// TIA Portal V17 export
// export: Created 2025-03-05T08:02:19.8399003Z, ExportSetting WithDefaults, DisplayName Totally Integrated Automation Portal, DisplayVersion V17 Update 8, DisplayName TIA Portal Openness, DisplayVersion V17 Update 8, DisplayName TIA Portal Version Control Interface, DisplayVersion V17, DisplayName SINAMICS Startdrive Advanced, DisplayVersion V17 SP2, DisplayName SINAMICS Startdrive G110M, G120, G120C, G120D, G120P, G115D, DisplayVersion V17 SP2, DisplayName SINAMICS Startdrive G130, G150, S120, S150, SINAMICS MV, S210, DisplayVersion V17 SP2, DisplayName STEP 7 Professional, DisplayVersion V17 Update 8, DisplayName SINUMERIK ONE STEP 7 Toolbox, DisplayVersion V17 Update 12, DisplayName SINUMERIK 840D sl STEP 7 Toolbox, DisplayVersion V17 Update 12, DisplayName STEP 7 Safety, DisplayVersion V17 Update 6, DisplayName WinCC Advanced, DisplayVersion V17 Update 8
TYPE "AXIS_MANAGEMENT"
// stored: IsFailsafeCompliant false
   STRUCT
      UNIT_01_HM_PSTN : Bool;   // UNIT 01 HOME POSITION
      UNIT_01_MAINT_POS : Bool;   // UNIT 01 MAINTENACE POSITION
      UNIT_01_ST1_OUT_OF_CLLSN_ST0 : Bool;   // UNIT 01 STATION 1 OUT OF COLLISION STATION 0
      UNIT_01_ST2_OUT_OF_CLLSN_ST0 : Bool;   // UNIT 01 STATION 2 OUT OF COLLISION STATION 0
      UNIT_01_ST3_OUT_OF_CLLSN_ST0 : Bool;   // UNIT 01 STATION 3 OUT OF COLLISION STATION 0
      UNIT_01_ST4_OUT_OF_CLLSN_ST0 : Bool;   // UNIT 01 STATION 4 OUT OF COLLISION STATION 0
      UNIT_01_ST3_AX_IN_HM_PSTN_XYZ : Bool;   // UNIT 01 STATION 3 AXIS IN HOME POSITION X-Y-Z
      UNIT_01_SPINDLES_STOP_AUX : Bool;   // UNIT 01 SPINDLES STOPPED AUXILIARY
      UNIT_01_MRPS_P_GG_RTN : Bool;   // UNIT 01 MARPOSS PLUG GAUGE RETURNED
      UNIT_01_IN_TL_POS : Bool;   // UNIT 01 IN TOOL POSITION
      UNIT_02_HM_PSTN : Bool;   // UNIT 02 HOME POSITION
      UNIT_02_MAINT_POS : Bool;   // UNIT 02 MAINTENACE POSITION
      UNIT_02_ST1_OUT_OF_CLLSN_ST0 : Bool;   // UNIT 02 STATION 1 OUT OF COLLISION STATION 0
      UNIT_02_ST2_OUT_OF_CLLSN_ST0 : Bool;   // UNIT 02 STATION 2 OUT OF COLLISION STATION 0
      UNIT_02_ST3_OUT_OF_CLLSN_ST0 : Bool;   // UNIT 02 STATION 3 OUT OF COLLISION STATION 0
      UNIT_02_ST4_OUT_OF_CLLSN_ST0 : Bool;   // UNIT 01 STATION 4 OUT OF COLLISION STATION 0
      UNIT_02_ST3_AX_IN_HM_PSTN_XYZ : Bool;   // UNIT 02 AXIS IN HOME POSITION X-Y-Z
      UNIT_02_SPINDLES_STOP_AUX : Bool;   // UNIT 02 SPINDLES STOPPED AUXILIARY
      UNIT_02_MRPSS_MSRG_PRB_RTN : Bool;   // UNIT 02 MARPOSS PLUG GAUGE RETURNED
      UNIT_02_IN_TL_POS : Bool;   // UNIT 02 IN TOOL POSITION
      UNIT_01_ST0_AX_E10_HM_PSTN : Bool;   // UNIT 01 STATION 0 AXIS E10 HOME POSITION
      UNIT_02_ST0_AX_E20_HM_PSTN : Bool;   // UNIT 02 STATION 0 AXIS E20 HOME POSITION
      FIXTURE_HM_PSTN : Bool;   // UNIT FIXTURE HOME POSITION
      FIXTURE_DBB70_0 : Bool;   // UNIT FIXTURE DBB70=0 (90)
      FIXTURE_DBB70_1 : Bool;   // UNIT FIXTURE DBB70=1 (-90)
      FIXTURE_1_LOAD_UNLOAD_POS : Bool;   // FIXTURE 1 IN LOAD UNLOAD POSITION (180)
      FIXTURE_2_LOAD_UNLOAD_POS : Bool;   // FIXTURE 2 IN LOAD UNLOAD POSITION (0)
      FIXTURE_1_MANUAL_LOAD_UNLOAD_POS : Bool;   // FIXTURE 1 IN MANUAL LOAD UNLOAD POSITION
      FIXTURE_2_MANUAL_LOAD_UNLOAD_POS : Bool;   // FIXTURE 2 IN MANUAL LOAD UNLOAD POSITION
      GENRL_RTN_CND_ALL_CLG_CYL_UNIT_01 : Bool;   // GENERAL RETURN CONDITIONS FOR ALL CLAMPING CYLINDERS UNIT 01
      GENRL_RTN_CND_ALL_CLG_CYL_UNIT_02 : Bool;   // GENERAL RETURN CONDITIONS FOR ALL CLAMPING CYLINDERS UNIT 02
      CH1_PRMR_SET_SLCTN_A : Bool;   // CHANNEL 1 PARAMETER SET SELECTION A
      CH2_PRMR_SET_SLCTN_A : Bool;   // CHANNEL 2 PARAMETER SET SELECTION A
      CH3_PRMR_SET_SLCTN_A : Bool;   // CHANNEL 3 PARAMETER SET SELECTION A
      CH4_PRMR_SET_SLCTN_A : Bool;   // CHANNEL 4 PARAMETER SET SELECTION A
      CH5_PRMR_SET_SLCTN_A : Bool;   // CHANNEL 5 PARAMETER SET SELECTION A
      CH6_PRMR_SET_SLCTN_A : Bool;   // CHANNEL 6 PARAMETER SET SELECTION A
      CH7_PRMR_SET_SLCTN_A : Bool;   // CHANNEL 7 PARAMETER SET SELECTION A
      CH8_PRMR_SET_SLCTN_A : Bool;   // CHANNEL 8 PARAMETER SET SELECTION A
      CH9_PRMR_SET_SLCTN_A : Bool;   // CHANNEL 9 PARAMETER SET SELECTION A
      CH10_PRMR_SET_SLCTN_A : Bool;   // CHANNEL 10 PARAMETER SET SELECTION A
      CH1_PRMR_SET_SLCTD_A : Bool;   // CHANNEL 1 PARAMETER SET SELECTED A
      CH2_PRMR_SET_SLCTD_A : Bool;   // CHANNEL 2 PARAMETER SET SELECTED A
      CH3_PRMR_SET_SLCTD_A : Bool;   // CHANNEL 3 PARAMETER SET SELECTED A
      CH4_PRMR_SET_SLCTD_A : Bool;   // CHANNEL 4 PARAMETER SET SELECTED A
      CH5_PRMR_SET_SLCTD_A : Bool;   // CHANNEL 5 PARAMETER SET SELECTED A
      CH6_PRMR_SET_SLCTD_A : Bool;   // CHANNEL 6 PARAMETER SET SELECTED A
      CH7_PRMR_SET_SLCTD_A : Bool;   // CHANNEL 7 PARAMETER SET SELECTED A
      CH8_PRMR_SET_SLCTD_A : Bool;   // CHANNEL 8 PARAMETER SET SELECTED A
      CH9_PRMR_SET_SLCTD_A : Bool;   // CHANNEL 9 PARAMETER SET SELECTED A
      CH10_PRMR_SET_SLCTD_A : Bool;   // CHANNEL 10 PARAMETER SET SELECTED A
   END_STRUCT;
END_TYPE
